Fanuc TP program (LS listing): MOVE_HOME.LS

/PROG  MOVE_HOME
/ATTR
OWNER		= MNEDITOR;
COMMENT		= "";
PROG_SIZE	= 207;
CREATE		= DATE 18-04-05  TIME 10:27:12;
MODIFIED	= DATE 18-04-05  TIME 10:27:20;
FILE_NAME	= ;
VERSION		= 0;
LINE_COUNT	= 1;
MEMORY_SIZE	= 575;
PROTECT		= READ_WRITE;
TCD:  STACK_SIZE	= 0,
      TASK_PRIORITY	= 50,
      TIME_SLICE	= 0,
      BUSY_LAMP_OFF	= 0,
      ABORT_REQUEST	= 0,
      PAUSE_REQUEST	= 0;
DEFAULT_GROUP	= 1,*,*,*,*;
CONTROL_CODE	= 00000000 00000000;
/APPL

AUTO_SINGULARITY_HEADER;
  ENABLE_SINGULARITY_AVOIDANCE   : TRUE;

  AUTOZONE_INTERFERENCE_AVOID;
    AUTOZONE_ENABLED         : FALSE;
    AUTOZONE_SCHEDULE_NUMBER : 1;
/MN
   1:J PR[1:HOME] 3% FINE    ;
/POS
/END
